Staubli VAL3: Entwicklungsmethodik.pjx

--- Entwicklungsmethodik.pjx ---
Parameters version=s8.3.1Cs9_BS885 stackSize=100000 millimeterUnit=true
Program file=pick.pgx
Program file=PickPlace.pgx
Program file=place.pgx
Program file=start.pgx
Program file=stop.pgx
Program file=TCPserver.pgx
Program file=Vereinzeln.pgx
Data file=Entwicklungsmethodik.dtx

--- Entwicklungsmethodik.dtx ---
mdesc mNomSpeed
frame fUserFrame = {x=1007.262395, y=-312.843264, z=-186.866453, rx=-0.535332, ry=-0.21904, rz=90.124968, fatherId=world[0]}
sio soTcpClient = {link=Socket\server0}
jointRx jHome = {j3=90, j5=90}
bool bNewData
num nData[5]
bool bReady
tool tGreiferM = {y=-27, z=127, rx=45, fatherId=flange[0], ioLink=ValveIO\valve1, ioOpen=0.05, ioClose=0.05}
tool tGreiferS = {y=27, z=127, rx=-45, ry=5.50371872946114E-07, rz=179.999999432294, fatherId=flange[0], ioLink=ValveIO\valve1, ioOpen=0.05, ioClose=0.05}
bool bVereinzeln
bool bPick
trsf trApro = {z=-150}
pointRx pPick[4]
  [0] = {z=6, rx=180, rz=45, fatherId=fUserFrame[0]}
  [1] = {z=20, rx=180, rz=45, fatherId=fUserFrame[0]}
  [2] = {z=6, rx=180, rz=45, fatherId=fUserFrame[0]}
  [3] = {z=10, rx=180, rz=45, fatherId=fUserFrame[0]}
mdesc mUsedSpeed
pointRx pPlace = {z=50, rx=180, rz=45, fatherId=fUserFrame[0]}
num nObj
num nOrientation
num nX
num nY
num nAngle
pointRx pVereinzeln = {z=10, rx=180, rz=45, fatherId=fUserFrame[0]}
trsf trVer = {x=100}
mdesc mVereinzeln = {accel=10, leave=1, reach=1}
num nX_S
num nX_M
num nY_M
num nY_S
dio delta_Y
dio delta_X
pointRx pEmpty = {fatherId=fUserFrame[0]}
jointRx jEmpty
pointRx pObj[10]
  [0] = {x=345, y=445, rz=350, fatherId=fUserFrame[0]}
  [1] = {x=256, y=423, rz=348, fatherId=fUserFrame[0]}
  [2] = {x=144, y=415, rz=354, fatherId=fUserFrame[0]}
  [3] = {x=71, y=410, rz=323, fatherId=fUserFrame[0]}
  [4] = {x=449, y=370, rz=224, fatherId=fUserFrame[0]}
  [5] = {x=163, y=356, rz=335, fatherId=fUserFrame[0]}
  [6] = {x=347, y=337, rz=182, fatherId=fUserFrame[0]}
  [7] = {x=84, y=333, rz=333, fatherId=fUserFrame[0]}
  [8] = {x=263, y=246, rz=523, fatherId=fUserFrame[0]}
  [9] = {x=406, y=235, rz=511, fatherId=fUserFrame[0]}
pointRx pAblegen[2]
  [0] = {x=700, y=125, fatherId=fUserFrame[0]}
  [1] = {x=700, y=375, fatherId=fUserFrame[0]}

--- start.pgx ---
program start()
begin

  clearBuffer(soTcpClient)
  movej(jHome,tGreiferM,mUsedSpeed)


  taskCreate "TCP-Server", 10, TCPserver()

  taskCreate "p&p", 5, PickPlace()

  taskCreate "Vereinzeln", 5, Vereinzeln()



  movej(jHome,tGreiferM,mUsedSpeed)
  waitEndMove()

end

--- pick.pgx ---
program pick(num x_nX, num x_nY, num x_angle, tool tGreifer)
  local num i
begin

  i = 0


  switch nData[0]

    case 1
      if nData[1] == 1
        i = 1
      endIf

    break
    case 2
      if nData[1] == 1
        i = 3
      else
        i = 2
      endIf


    break
    default
      i = 1
    break
  endSwitch

  logMsg("n_Y "+toString(".4",x_nY))
  //logMsg("i: " + toString("0.4",i))
  pPick[i].trsf.x = x_nX
  pPick[i].trsf.y = x_nY
  pPick[i].trsf.rz = x_angle



  movej(appro(pPick[i],trApro),tGreifer, mUsedSpeed)
  movel(pPick[i], tGreifer, mUsedSpeed)
  close(tGreifer)
  movel(appro(pPick[i], trApro), tGreifer, mUsedSpeed)
  logMsg("Objekt aufgegriffen")







end

--- PickPlace.pgx ---
program PickPlace()
  local tool tGreifer
  local num x
  local num y
begin

  // initialisieren der KKs der Ablagestapel
  // delta_Y = 270
  //delta_X = 80

  nX_M = 650
  nY_M = 40


  nX_S = 650
  nY_S = 290

  x = 0
  y = 0


  while true


    // Greift Objekte auf und legt diese ab


    wait(bNewData)

    // Wenn wir nicht vereinzeln heben wir Obj auf und setzen diese ab
    if bVereinzeln
    else

      logMsg(" Pick Place startet")
      if nData[0]==1
        tGreifer = tGreiferM
        x = nX_M
        y = nY_M
      else
        tGreifer = tGreiferS
        x = nX_S
        y = nY_S
      endIf

      if bPick
        call pick(nX,nY,nAngle,tGreifer)
        call place(x,y,tGreifer)
      endIf


      // Ablagepositionen ändern

      switch nData[0]
        case 1
          nX_M = nX_M + 50

          if nX_M > 730
            nX_M = 650
            nY_M = nY_M + 50
          endIf


          if nY_M > 310
            nY_M = 310
            nX_M = 650+15
          endIf

        break

        case 2

          nX_S = nX_S + 40

          if nX_S > 730
            nX_S = 650
            nY_S = nY_S + 70
          endIf

          if nY_S > 560
            nY_S = 290
            nX_S = 650+15
          endIf


        break
      endSwitch




      // Return Value
      bNewData = false
      bReady = true



    endIf



  endWhile

end

--- place.pgx ---
program place(num x_nX, num x_nY, tool tGreifer)
begin
  // x,y [mm]


  pPlace.trsf.x = x_nX
  pPlace.trsf.y = x_nY



  movej(appro(pPlace,trApro),tGreifer, mUsedSpeed)
  movel(pPlace, tGreifer, mUsedSpeed)
  open(tGreifer)
  movel(appro(pPlace, trApro), tGreifer, mUsedSpeed)
  logMsg("Objekt abgelegt")





end

--- TCPserver.pgx ---
program TCPserver()
  local num l_nStatus
  local num l_nBytesIn[40]
  local num l_nSuccBytes
  local pointRx p_point
  local bool erreichbar
  local bool error
begin
  // l_nBytesIn: 64 bit -> 8 byte
  // nData: 8



  while true
    logMsg("Schleife start")
    l_nStatus=sioGet(soTcpClient, l_nBytesIn)
    if l_nStatus>0
      // Write recieved bytes in data
      // Achtung bei mehr Bitlänge 24, 3 und globale Variable(nData) ändern

      if(fromBinary(l_nBytesIn,40,"8.0l",nData)!=5)
        logMsg("Empfangene Daten sind fehlerhaft",2)

      else
        logMsg("Daten über TCP/IP empfangen")
        // check if data is in limits
        // ...
        nObj = limit(nData[0],1,10)
        nOrientation = limit(nData[1],1,2)
        nX = limit(nData[2],1,750)
        nY = limit(nData[3],1,500)
        nAngle = nData[4]
        // logMsg(toString(".4",nData[0]))
        //logMsg(toString(".4",nData[1]))
        //logMsg(toString(".4",nData[3]))
        //logMsg(toString(".4",nY))
        //logMsg(toString(".4",nData[3]))
        //logMsg(toString(".4",nData[4]))


        // check if the Point is reachable
        error = false
        pEmpty.trsf.x = nX
        pEmpty.trsf.y = nY
        pEmpty.trsf.z = 10
        pEmpty.trsf.rz = nAngle
        //
        if nData[0] == 3
          while !pointToJoint(tGreiferM,jHome,pEmpty,jEmpty)
            pEmpty.trsf.rz = pEmpty.trsf.rz + 5
            nAngle = pEmpty.trsf.rz
          endWhile
        endIf


        if !pointToJoint(tGreiferM,jHome,pEmpty,jEmpty)
          pEmpty.trsf.rz = nAngle + 180


          if pointToJoint(tGreiferM,jHome,pEmpty,jEmpty)
            nAngle = nAngle + 180
           // logMsg("Punkt wird verändert")
          else
            // logMsg("Punkt nicht erreichbar")

            error = true
          endIf

        endIf


        if error == false


          // if Vereinzeln ist True
          if nData[0]==3

            bPick = false
            bVereinzeln = true
          else
            bPick = true
            bVereinzeln = false
          endIf



          bReady = false
          bNewData = true

        else
          bReady = true
          logMsg(" ****************** Punkt ist nicht erreichbar!!")

        endIf

      endIf



      // tell client that robot is ready
      wait(bReady)

      //delay(2)
      l_nStatus=sioSet(soTcpClient, 1)
    endIf
  endWhile
end

--- Vereinzeln.pgx ---
program Vereinzeln()
  local mdesc mDesc
begin


  while true

    // Vereinzelt die Objekte


    wait(bNewData)

    // Wenn wir nicht vereinzeln heben wir Obj auf und setzen diese ab
    if bVereinzeln
      logMsg("Vereinzeln startet ")

      pVereinzeln.trsf.x = nX
      pVereinzeln.trsf.y = nY
      pVereinzeln.trsf.rz = nAngle


      logMsg("nAngle ****************** " + toString("0.4", nAngle))
      logMsg("nData ****************** " + toString("0.4", nData[4] ))
      close(tGreiferM)
      // Fahre über Punkt Vereinzeln --> irgenwie
      movej(appro(pVereinzeln, trApro), tGreiferM, mUsedSpeed)


      movej(pVereinzeln, tGreiferM, mVereinzeln)

      // Fahre linear trVer voraus
      pVereinzeln.trsf.x =  pVereinzeln.trsf.x +  100 * cos(-nData[4])
      pVereinzeln.trsf.y =  pVereinzeln.trsf.y +  100 * sin(-nData[4])

      movej(pVereinzeln,tGreiferM, mVereinzeln)
      // fahre vom letzten POSE appro(pVereinzeln,trVer) --> zur neuen oberhalb, --> trApro

      movej(appro(pVereinzeln, trApro), tGreiferM, mVereinzeln)


      logMsg("Objekt vereinzelt")

      // Return Value
      bNewData = false
      bReady = true


    endIf






  endWhile

end
